PROGRAM InitBitMasks
VAR
	nCounter : int;
END_VAR

FOR nCounter:=1 TO 32 BY 1 DO
	bitMasks[nCounter] := SHL(16#1,nCounter);
END_FOR

END_PROGRAM

(* stored: Version 1.1.0.1, ProductVersion 3.1.4020.12
   POU InitBitMasks: Id {ec4f62a5-cd2f-4f9b-9760-127006f90bc0}, SpecialFunc None *)
